// TwinCAT 3 PLC project PLC1
// ProgramVersion: 3.1.4024.12
// libraries:
//   Tc2_Standard, * (Beckhoff Automation GmbH)
//   Tc2_System, * (Beckhoff Automation GmbH)
//   Tc2_Utilities, * (Beckhoff Automation GmbH)
//   Tc3_Module, * (Beckhoff Automation GmbH)
// project tree:
//   DUTs/ ST_DUT.TcDUT
//   / PlcTask.TcTTO
//   POUs/ MAIN.TcPOU, SavePV.TcPOU
// real-time tasks:
//   TASK PlcTask: cycle T#10ms, priority 20, ADS port 350

CONFIGURATION PLC1
    RESOURCE PLC ON TwinCAT3
        TASK PlcTask(INTERVAL := T#10ms, PRIORITY := 20);
        PROGRAM MAIN WITH PlcTask : MAIN;
    END_RESOURCE
END_CONFIGURATION

// ---- DUTs/ST_DUT.TcDUT
TYPE ST_DUT :
STRUCT
	sFirstName	:	STRING;
	sLastName	:	STRING;
	sUserName	:	STRING;
	iPin		:	UINT;
	sDateCreated:	STRING;
	bAdmin		:	BOOL;
	bDisable	:	BOOL;
END_STRUCT
END_TYPE

// ---- POUs/MAIN.TcPOU
PROGRAM MAIN
VAR PERSISTENT 
    aArray : ARRAY[0..24] OF ST_DUT;
END_VAR 

VAR
	iSelectedRow : UINT;
	bDeleteRow : BOOL;
	bConsolidate: BOOL;
	iConsolCount : UINT;
	bEmpty: BOOL;
	iEmptyCount : UINT;
END_VAR

SavePV();

IF bDeleteRow THEN
	aArray[iSelectedRow].sFirstName := '';
	aArray[iSelectedRow].sLastName := '';
	aArray[iSelectedRow].sUserName := '';
	aArray[iSelectedRow].iPin := 0;
	aArray[iSelectedRow].sDateCreated := '';
	aArray[iSelectedRow].bAdmin := FALSE;
	aArray[iSelectedRow].bDisable := FALSE;
	bDeleteRow := FALSE;
	bConsolidate := TRUE;
END_IF

IF bEmpty THEN
	FOR iEmptyCount := 0 TO 24 DO
		aArray[iEmptyCount].sFirstName := '';
		aArray[iEmptyCount].sLastName := '';
		aArray[iEmptyCount].sUserName := '';
		aArray[iEmptyCount].sDateCreated := '';
		aArray[iEmptyCount].iPin := 0;
		aArray[iEmptyCount].bAdmin := FALSE;
		aArray[iEmptyCount].bDisable := FALSE;
	END_FOR
	bEmpty := FALSE;
END_IF


IF bConsolidate THEN
	FOR iConsolCount := 0 TO 24 DO
		IF aArray[iConsolCount].sFirstName = '' THEN
			aArray[iConsolCount] := aArray[iConsolCount + 1];
		END_IF
		IF aArray[iConsolCount].sFirstName = aArray[iConsolCount + 1].sFirstName THEN
			aArray[iConsolCount + 1].sFirstName := '';
			aArray[iConsolCount + 1].sLastName := '';
			aArray[iConsolCount + 1].sUserName := '';
			aArray[iConsolCount + 1].sDateCreated := '';
			aArray[iConsolCount + 1].iPin := 0;
			aArray[iConsolCount + 1].bAdmin := FALSE;
			aArray[iConsolCount + 1].bDisable := FALSE;
		END_IF
	END_FOR
	bConsolidate := FALSE;
END_IF

END_PROGRAM

// ---- POUs/SavePV.TcPOU
PROGRAM SavePV
VAR
	fbWritePersistent		:		WritePersistentData;
	TonStart				:		TON;
	TonInterval				:		TON;
	r_trigStart				:		R_TRIG;
	bStartWrite				:		BOOL;
	bWriteNow				:		BOOL;
END_VAR

//Backup the machine config vars
//Write a backup when the machine starts - on rising edge
	r_trigStart(CLK:= TonStart.Q);
	TonStart(IN:= TRUE, PT:= T#10MS);

//backup persistent vars every 1 minute
	TonInterval(IN:=TonStart.Q AND NOT fbWritePersistent.BUSY, PT:= T#60S);

	fbWritePersistent(
		NETID:= '', 
		PORT:= 851, 
		START:= bStartWrite, 
		TMOUT:= T#10S);
		
//Execute the backup
	IF NOT fbWritePersistent.Busy AND r_trigStart.Q THEN
		bStartWrite := TRUE;
	ELSIF NOT fbWritePersistent.BUSY AND TonInterval.Q THEN
		bStartWrite := TRUE;
	ELSIF NOT fbWritePersistent.BUSY AND bWriteNow THEN
		bStartWrite := TRUE;
	ELSE
		bStartWrite := FALSE;
	END_IF

END_PROGRAM
